% RSLogix 500 project INTRO TO PLC JOB HO4 ADAM REISKE.RSS, saved by version 10.00.00.00 %
PROJECT "UNTITLED"    % processor: Bul.1763 MicroLogix 1100 Series B %

PROGRAM FILES
  LAD 2   9 rungs

DATA FILES
  O0 OUTPUT  4 elements
  I1 INPUT  6 elements
  S2 STATUS  66 elements
  B3 BINARY  1 elements
  T4 TIMER  1 elements
  C5 COUNTER  1 elements
  R6 CONTROL  1 elements
  N7 INTEGER  1 elements
  F8 FLOAT  1 elements

LADDER 2
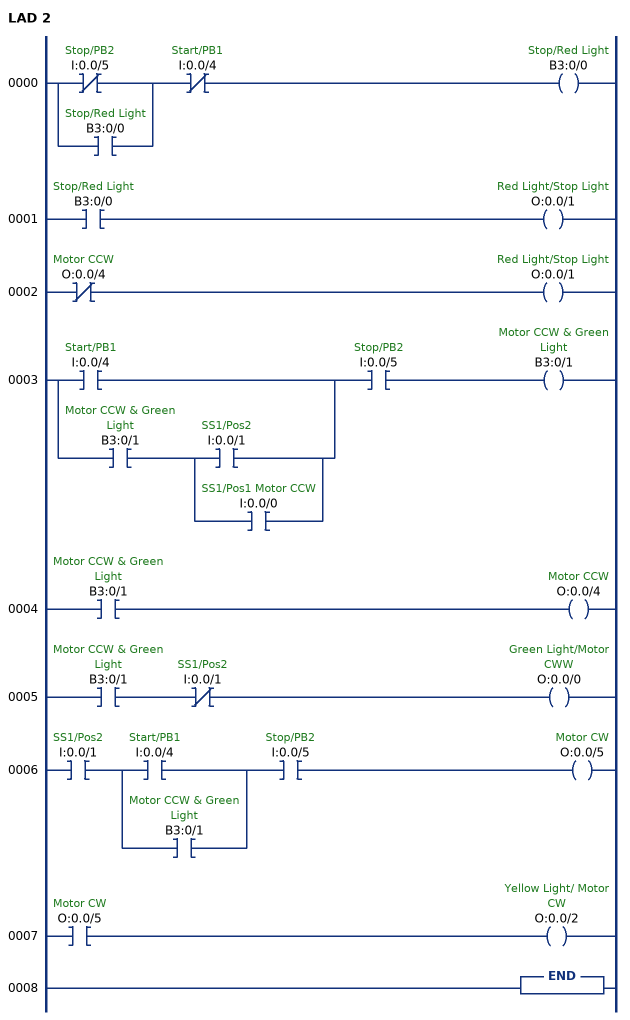
% Rung: 0 %
SOR BST XIO I:0.0/5 NXB XIC B3:0/0 BND XIO I:0.0/4 OTE B3:0/0 EOR
%   I:0.0/5  "Stop/PB2" %
%   B3:0/0  "Stop/Red Light" %
%   I:0.0/4  "Start/PB1" %
% Rung: 1 %
SOR XIC B3:0/0 OTE O:0.0/1 EOR
%   B3:0/0  "Stop/Red Light" %
%   O:0.0/1  "Red Light/Stop Light" %
% Rung: 2 %
SOR XIO O:0.0/4 OTE O:0.0/1 EOR
%   O:0.0/4  "Motor CCW" %
%   O:0.0/1  "Red Light/Stop Light" %
% Rung: 3 %
SOR BST XIC I:0.0/4 NXB XIC B3:0/1 BST XIC I:0.0/1 NXB XIC I:0.0/0 BND BND XIC I:0.0/5 OTE B3:0/1 EOR
%   I:0.0/4  "Start/PB1" %
%   B3:0/1  "Motor CCW & Green Light" %
%   I:0.0/1  "SS1/Pos2" %
%   I:0.0/0  "SS1/Pos1 Motor CCW" %
%   I:0.0/5  "Stop/PB2" %
% Rung: 4 %
SOR XIC B3:0/1 OTE O:0.0/4 EOR
%   B3:0/1  "Motor CCW & Green Light" %
%   O:0.0/4  "Motor CCW" %
% Rung: 5 %
SOR XIC B3:0/1 XIO I:0.0/1 OTE O:0.0/0 EOR
%   B3:0/1  "Motor CCW & Green Light" %
%   I:0.0/1  "SS1/Pos2" %
%   O:0.0/0  "Green Light/Motor CWW" %
% Rung: 6 %
SOR XIC I:0.0/1 BST XIC I:0.0/4 NXB XIC B3:0/1 BND XIC I:0.0/5 OTE O:0.0/5 EOR
%   I:0.0/1  "SS1/Pos2" %
%   I:0.0/4  "Start/PB1" %
%   B3:0/1  "Motor CCW & Green Light" %
%   I:0.0/5  "Stop/PB2" %
%   O:0.0/5  "Motor CW" %
% Rung: 7 %
SOR XIC O:0.0/5 OTE O:0.0/2 EOR
%   O:0.0/5  "Motor CW" %
%   O:0.0/2  "Yellow Light/ Motor CW" %
% Rung: 8 %
SOR END EOR

OTHER DOCUMENTED ADDRESSES
  B3:0/2  "stop"
  B3:0/3  "STOP"
  B3:0/4  B
